FUNCTION_BLOCK Decode1to5 (* Basic FB with empty ECC *)
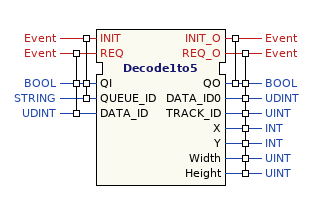
  EVENT_INPUT
    INIT WITH QUEUE_ID, QI;
    REQ WITH QI, DATA_ID;
  END_EVENT
  EVENT_OUTPUT
    INIT_O WITH QO;
    REQ_O WITH QO, Height, Width, Y, X, TRACK_ID, DATA_ID0;
  END_EVENT
  VAR_INPUT
    QI : BOOL;
    QUEUE_ID : STRING;
    DATA_ID : UDINT;
  END_VAR
  VAR_OUTPUT
    QO : BOOL;
    DATA_ID0 : UDINT;
    TRACK_ID : UINT;
    X : INT;
    Y : INT;
    Width : UINT;
    Height : UINT;
  END_VAR
END_FUNCTION_BLOCK
